KUKA KRL program: GetMillingRPM.src

&ACCESS RV1
&PARAM EDITMASK = *
DEFFCT REAL GetMillingRPM(lrCuttingSpeed :IN,lrMillingToolDiameter :IN)
REAL lrCuttingSpeed
REAL lrMillingToolDiameter

  RETURN (lrCuttingSpeed*1000)/(3.14*lrMillingToolDiameter)

ENDFCT
